FUNCTION_BLOCK OthersDishcargeValvesBasic (* Basic Function Block Type *)
  (* Standard: 61499-2 *)
  (* Version 0.0, 11/29/2023, SESA371406, Schneider Electric, Template *)
  PACKAGE SE.Nereda;
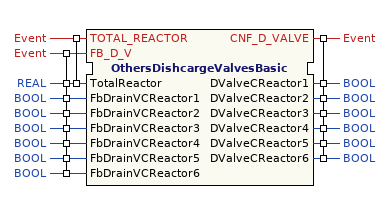
  EVENT_INPUT
    TOTAL_REACTOR WITH TotalReactor; (* Normal Execution Request *)
    FB_D_V WITH FbDrainVCReactor1, FbDrainVCReactor2, FbDrainVCReactor3, FbDrainVCReactor4, FbDrainVCReactor5, FbDrainVCReactor6, TotalReactor;
  END_EVENT
  EVENT_OUTPUT
    CNF_D_VALVE WITH DValveCReactor1, DValveCReactor4, DValveCReactor5, DValveCReactor6, DValveCReactor2, DValveCReactor3; (* Execution Confirmation *)
  END_EVENT
  VAR_INPUT
    TotalReactor : REAL; (* Input event qualifier *)
    FbDrainVCReactor1 : BOOL;
    FbDrainVCReactor2 : BOOL;
    FbDrainVCReactor3 : BOOL;
    FbDrainVCReactor4 : BOOL;
    FbDrainVCReactor5 : BOOL;
    FbDrainVCReactor6 : BOOL;
  END_VAR
  VAR_OUTPUT
    DValveCReactor1 : BOOL; (* Output event qualifier *)
    DValveCReactor2 : BOOL;
    DValveCReactor3 : BOOL;
    DValveCReactor4 : BOOL;
    DValveCReactor5 : BOOL;
    DValveCReactor6 : BOOL;
  END_VAR
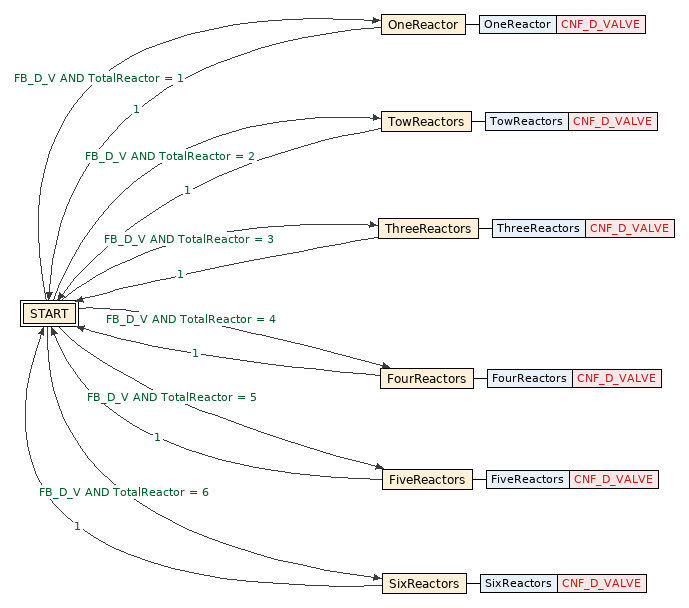
  EC_STATES
    START; (* Initial State *)
    OneReactor : OneReactor -> CNF_D_VALVE;
    TowReactors : TowReactors -> CNF_D_VALVE;
    ThreeReactors : ThreeReactors -> CNF_D_VALVE;
    FourReactors : FourReactors -> CNF_D_VALVE;
    FiveReactors : FiveReactors -> CNF_D_VALVE;
    SixReactors : SixReactors -> CNF_D_VALVE;
  END_STATES
  EC_TRANSITIONS
    START TO OneReactor := FB_D_V AND TotalReactor = 1;
    OneReactor TO START := 1;
    START TO TowReactors := FB_D_V AND TotalReactor = 2;
    TowReactors TO START := 1;
    START TO ThreeReactors := FB_D_V AND TotalReactor = 3;
    ThreeReactors TO START := 1;
    START TO FourReactors := FB_D_V AND TotalReactor = 4;
    FourReactors TO START := 1;
    START TO FiveReactors := FB_D_V AND TotalReactor = 5;
    FiveReactors TO START := 1;
    START TO SixReactors := FB_D_V AND TotalReactor = 6;
    SixReactors TO START := 1;
  END_TRANSITIONS
  ALGORITHM OneReactor IN ST:
;
DValveCReactor1 := TRUE;
DValveCReactor2 := FALSE;
DValveCReactor3 := FALSE;
DValveCReactor4 := FALSE;
DValveCReactor5 := FALSE;
DValveCReactor6 := FALSE;
  END_ALGORITHM
  ALGORITHM TowReactors IN ST:
;
//Operating condition Reacotr1:
IF FbDrainVCReactor1 THEN
	DValveCReactor2 := TRUE;
ELSE
	DValveCReactor2 := FALSE;
END_IF;

//Operating condition Reacotr2:
IF FbDrainVCReactor2 THEN
	DValveCReactor1 := TRUE;
ELSE
	DValveCReactor1 := FALSE;
END_IF;
  END_ALGORITHM
  ALGORITHM ThreeReactors IN ST:
;
// Operating condition Reactor 1:
IF FbDrainVCReactor2 AND FbDrainVCReactor3 THEN
	DValveCReactor1 := TRUE;
ELSE
	DValveCReactor1 := FALSE;
END_IF;


// Operating condition Reactor 2:
IF FbDrainVCReactor1 AND FbDrainVCReactor3 THEN
	DValveCReactor2 := TRUE;
ELSE
	DValveCReactor2 := FALSE;
END_IF;


// Operating condition Reactor 3:
IF FbDrainVCReactor1 AND FbDrainVCReactor2 THEN
	DValveCReactor3 := TRUE;
ELSE
	DValveCReactor3 := FALSE;
END_IF;
  END_ALGORITHM
  ALGORITHM FourReactors IN ST:
;
// Operating condition Reactor 1:
IF FbDrainVCReactor2 AND FbDrainVCReactor3 AND FbDrainVCReactor4 THEN
	DValveCReactor1 := TRUE;
ELSE
	DValveCReactor1 := FALSE;
END_IF;


// Operating condition Reactor 2:
IF FbDrainVCReactor1 AND FbDrainVCReactor3 AND FbDrainVCReactor4 THEN
	DValveCReactor2 := TRUE;
ELSE
	DValveCReactor2 := FALSE;
END_IF;


// Operating condition Reactor 3:
IF FbDrainVCReactor1 AND FbDrainVCReactor2 AND FbDrainVCReactor4 THEN
	DValveCReactor3 := TRUE;
ELSE
	DValveCReactor3 := FALSE;
END_IF;


// Operating condition Reactor 4:
IF FbDrainVCReactor1 AND FbDrainVCReactor2 AND FbDrainVCReactor3 THEN
	DValveCReactor4 := TRUE;
ELSE
	DValveCReactor4 := FALSE;
END_IF;
  END_ALGORITHM
  ALGORITHM FiveReactors IN ST:
;
// Operating condition Reactor 1:
IF FbDrainVCReactor2 AND FbDrainVCReactor3 AND FbDrainVCReactor4 AND FbDrainVCReactor5 THEN
	DValveCReactor1 := TRUE;
ELSE
	DValveCReactor1 := FALSE;
END_IF;


// Operating condition Reactor 2:
IF FbDrainVCReactor1 AND FbDrainVCReactor3 AND FbDrainVCReactor4 AND FbDrainVCReactor5 THEN
	DValveCReactor2 := TRUE;
ELSE
	DValveCReactor2 := FALSE;
END_IF;


// Operating condition Reactor 3:
IF FbDrainVCReactor1 AND FbDrainVCReactor2 AND FbDrainVCReactor4 AND FbDrainVCReactor5 THEN
	DValveCReactor3 := TRUE;
ELSE
	DValveCReactor3 := FALSE;
END_IF;


// Operating condition Reactor 4:
IF FbDrainVCReactor1 AND FbDrainVCReactor2 AND FbDrainVCReactor3 AND FbDrainVCReactor5 THEN
	DValveCReactor4 := TRUE;
ELSE
	DValveCReactor4 := FALSE;
END_IF;


// Operating condition Reactor 5:
IF FbDrainVCReactor1 AND FbDrainVCReactor2 AND FbDrainVCReactor3 AND FbDrainVCReactor4 THEN
	DValveCReactor5 := TRUE;
ELSE
	DValveCReactor5 := FALSE;
END_IF;
  END_ALGORITHM
  ALGORITHM SixReactors IN ST:
;
// Operating condition Reactor 1:
IF FbDrainVCReactor2 AND FbDrainVCReactor3 AND FbDrainVCReactor4 AND FbDrainVCReactor5 AND FbDrainVCReactor6 THEN
	DValveCReactor1 := TRUE;
ELSE
	DValveCReactor1 := FALSE;
END_IF;


// Operating condition Reactor 2:
IF FbDrainVCReactor1 AND FbDrainVCReactor3 AND FbDrainVCReactor4 AND FbDrainVCReactor5 AND FbDrainVCReactor6 THEN
	DValveCReactor2 := TRUE;
ELSE
	DValveCReactor2 := FALSE;
END_IF;


// Operating condition Reactor 3:
IF FbDrainVCReactor1 AND FbDrainVCReactor2 AND FbDrainVCReactor4 AND FbDrainVCReactor5 AND FbDrainVCReactor6 THEN
	DValveCReactor3 := TRUE;
ELSE
	DValveCReactor3 := FALSE;
END_IF;


// Operating condition Reactor 4:
IF FbDrainVCReactor1 AND FbDrainVCReactor2 AND FbDrainVCReactor3 AND FbDrainVCReactor5 AND FbDrainVCReactor6 THEN
	DValveCReactor4 := TRUE;
ELSE
	DValveCReactor4 := FALSE;
END_IF;


// Operating condition Reactor 5:
IF FbDrainVCReactor1 AND FbDrainVCReactor2 AND FbDrainVCReactor3 AND FbDrainVCReactor4 AND FbDrainVCReactor6 THEN
	DValveCReactor5 := TRUE;
ELSE
	DValveCReactor5 := FALSE;
END_IF;


// Operating condition Reactor 6:
IF FbDrainVCReactor1 AND FbDrainVCReactor2 AND FbDrainVCReactor3 AND FbDrainVCReactor4 AND FbDrainVCReactor5 THEN
	DValveCReactor6 := TRUE;
ELSE
	DValveCReactor6 := FALSE;
END_IF;
  END_ALGORITHM
END_FUNCTION_BLOCK
